# EPICS autosave request: OxInstIPS/OxInstIPS_settings.req
$(P):DISABLE
$(P):SET:ACTIVITY
$(P):SET:CONTROL
$(P):SET:CURRENTSWEEPRATE
$(P):SET:FIELDSWEEPRATE
$(P):SET:REMOTE
$(P):SET:SETPOINTCURRENT
$(P):SET:SETPOINTFIELD
$(P):SET:SWEEPMODE:TYPE
$(P):SET:SWEEPMODE:UNITS
$(P):SET:UNLOCKED
